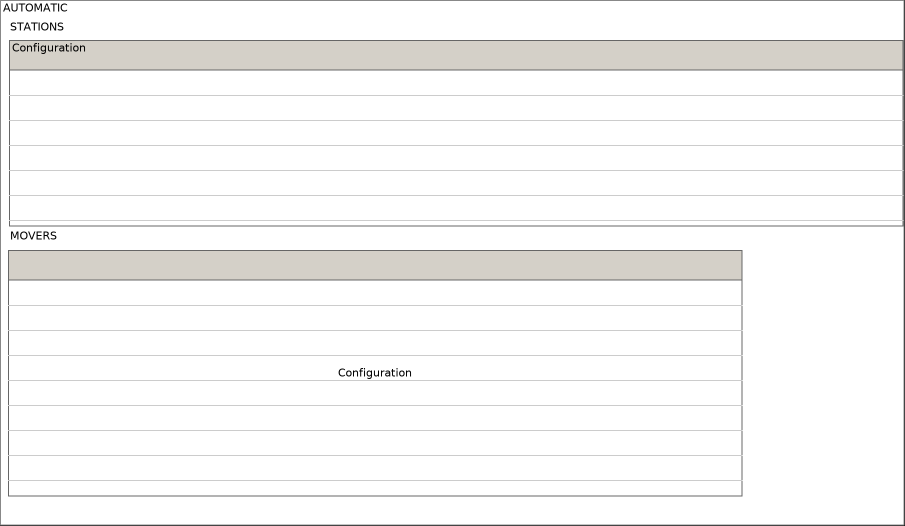
VISUALIZATION VI_XTSAutoVisu  // 905x526
VAR_IN_OUT
	xts : XTS_System;
END_VAR
VAR
	stTableStruct : ARRAY [1..25] OF stTableStructx10;
END_VAR
    Rectangle (0,0 905x526), "AUTOMATIC"
    Label (7,19 151x31), "STATIONS"
    Label (7,228 151x31), "MOVERS"
    Table (9,40 894x186), "Configuration", data array: stTableStruct
        p3854506369: xts.stCfg.stStationsCfg[INDEX].sName
        p1892666644: xts.stCfg.stStationsCfg[INDEX].bEnableManualAck
        p338671338: xts.stCfg.stStationsCfg[INDEX].bManualAck
        p2170511999: xts.aStations[INDEX].fbMoversFIFO.nMovers
        p3723444502: xts.aStations[INDEX].udiSequenceState
        p1218418051: xts.aStations[INDEX].udiErrorID
        p746581629: xts.aStations[INDEX].sMoversWaiting
        p3104783080: xts.aStations[INDEX].sMoversIn
        p2501879983: xts.aStations[INDEX].lrActualProcessTime
        p7306298: xts.aStations[INDEX].lrActualWaitingTime
        p511219082: M. Ack
        p4092479075: Movers Waiting
        p505689113: Error ID
        p4088588272: Movers In
        p2243050616: Process Time
        p516019884: Waiting Time
        p2685023577: stTableStruct.b1
        p3312258591: stTableStruct.b2
        p1791247317: stTableStruct.b3
        p262371475: stTableStruct.b4
        p4008173056: stTableStruct.b5
        p2340480326: stTableStruct.b6
        p606709900: stTableStruct.b7
        p1095668682: stTableStruct.b8
        p1037165547: stTableStruct.b9
        p1488378029: stTableStruct.b10
        Columns.Column.[9].Template: OnMouseClick: write the text variable via Default
        Columns.Column.[6].Template: OnMouseClick: write the text variable via Default, min 1, max 3
        Columns.Column.[4].Template: OnMouseClick: write the text variable via Default
        Columns.Column.[5].Template: OnMouseClick: write the text variable via Default
        Columns.Column.[2].Template: tap xts.stCfg.stStationsCfg[INDEX].bManualAck
        Columns.Column.[0].Template: OnMouseClick: write the text variable via Default
        Columns.Column.[7].Template: OnMouseClick: write the text variable via Default
        Columns.Column.[1].Template: toggle xts.stCfg.stStationsCfg[INDEX].bEnableManualAck
    Table (8,250 734x246), "Configuration", data array: stTableStruct
        p3854506369: xts.ax[INDEX].ax.NcToPlc.AxisId
        p1892666644: xts.ax[INDEX].ax.NcToPlc.ModuloSetPos
        p338671338: xts.ax[INDEX].ax.NcToPlc.SetVelo
        p2170511999: xts.ax[INDEX].ax.Status.MotionState
        p3723444502: xts.ax[INDEX].ax.NcToPlc.ErrorCode
        p2232123230: Name
        p511219082: Position
        p1755163831: Velocity
        p2237128397: Error ID
        p505689113: Process Time
        p1757482276: Stop Positions
        p4088588272: Ack Mode
        p2243050616: Disable
        p516019884: Travel Time
        p2685023577: stTableStruct.b1
        p3312258591: stTableStruct.b2
        p1791247317: stTableStruct.b3
        p262371475: stTableStruct.b4
        p4008173056: stTableStruct.b5
        p2340480326: stTableStruct.b6
        p606709900: stTableStruct.b7
        p1095668682: stTableStruct.b8
        p1037165547: stTableStruct.b9
        p1488378029: stTableStruct.b10
        Columns.Column.[6].Template: OnMouseClick: write the text variable via Default, min 1, max 3
        Columns.Column.[3].Template: OnMouseClick: write the text variable via Default
        Columns.Column.[8].Template: xts.aStations[INDEX].stCfg.bDisable=true; toggle xts.aStations[INDEX].stCfg.bDisable
        Columns.Column.[4].Template: OnMouseClick: write the text variable via Default
        Columns.Column.[5].Template: OnMouseClick: write the text variable via Default
        Columns.Column.[0].Template: OnMouseClick: OpenDialog Dialog=Mover_VISU, Parameters={fbMover: xts.aMovers[INDEX]}, OpenModal=True, OpenCentered=True
        Columns.Column.[7].Template: OnMouseClick: write the text variable via Default
        Columns.Column.[9].Template: OnMouseClick: write the text variable via Default
END_VISUALIZATION

(* stored: Version 1.1.0.1, ProductVersion 3.1.4024.11
   Visu VI_XTSAutoVisu: Id {f9e20e03-8613-4e3e-8212-6b9c477a923d} *)
